TEXTLIST Mc_Alarms
  0 = 'Machine Alarm 0'
  1 = 'alarm 2'
  2 = 'alarm 3'
  3 = 'alarm 4'
   = ''
END_TEXTLIST

(* stored: Version 1.1.0.1, ProductVersion 3.1.4024.12
   TextList Mc_Alarms: Id {4f6bd7c1-9320-0f76-291a-b54c4f409ed3} *)
